(* PLC project SafeLOGIC-1, BrAutomation SafeDESIGNER  4.3.3.7 *)
(* stored: companyURL http://www.br-automation.com, creationDateTime Wed Jan 30 17:54:31 2019 *)

PROGRAM Main
  VAR  (* added by the conversion: wires and edge detectors of the diagram *)
    _AND_S30_OUT : BOOL;
    _AND_S44_OUT : BOOL;
  END_VAR

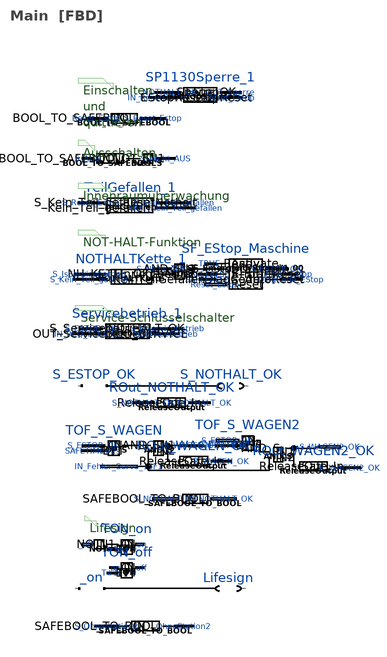
(* FBD diagram, written out as Structured Text *)
(* Einschalten und quittieren *)
SP1130Sperre_1(EStopOK := _NOTHALT_OK, EStopReset := IN_ResetNOTHALT);
Reset_Estop := SP1130Sperre_1.EStopReset2;
OUT_Sperre := SP1130Sperre_1.Sperre;
S_Reset_Estop := BOOL_TO_SAFEBOOL(Reset_Estop);
(* Ausschalten *)
S_Nicht_AUS := NOT_S(BOOL_TO_SAFEBOOL(S_AUS));
(* Innenraumüberwachung *)
TeilGefallen_1(S_ResetNothalt := S_Reset_Estop);
S_Kein_Teil_gefallen := TeilGefallen_1.S_Kein_Teil_gefallen;
OUT_Kein_Teil_gefallen := TeilGefallen_1.Kein_Teil_gefallen;
(* NOT-HALT-Funktion *)
NOTHALTKette_1(Einrichtbetrieb := S_IsServicebetrieb, KeinTeilGefallen := S_Kein_Teil_gefallen);
SF_EStop_Maschine(Activate := TRUE, S_EStopIn := AND_S(S_Nicht_AUS, NOTHALTKette_1.NH_KETTE_OK), S_StartReset := SAFEFALSE, S_AutoReset := SAFEFALSE, Reset := Reset_Estop);
S_ESTOP_OK := SF_EStop_Maschine.S_EStopOut;
DiagCode_EStop := SF_EStop_Maschine.DiagCode;
Error_Estop := SF_EStop_Maschine.Error;
(* Service-Schlüsselschalter *)
Servicebetrieb_1(NOTHALT_OK := S_ESTOP_OK, REQ_SERVICE := IN_REQ_SERVICE);
IsServicebetrieb := Servicebetrieb_1.OUT_Servicebetrieb;
S_IsServicebetrieb := Servicebetrieb_1.S_Servicebetrieb;
S_NOTHALT_OK := S_ESTOP_OK;
ROut_NOTHALT_OK(Safe_In := S_NOTHALT_OK);
R_NOTHALT_OK := ROut_NOTHALT_OK.ReleaseOut;
TOF_S_WAGEN(IN := S_ESTOP_OK, PT := SAFETIME#2s);
_AND_S30_OUT := AND_S(TOF_S_WAGEN.Q, IN_Fehler_Servo_15F1);
S_WAGEN_OK := _AND_S30_OUT;
TOF_S_WAGEN2(IN := S_ESTOP_OK, PT := SAFETIME#2s);
_AND_S44_OUT := AND_S(TOF_S_WAGEN2.Q, IN_Fehler_Servo_15F1);
S_WAGEN2_OK := _AND_S44_OUT;
ROut_WAGEN_OK(Safe_In := _AND_S30_OUT);
R_WAGEN_OK := ROut_WAGEN_OK.ReleaseOut;
ROut_WAGEN2_OK(Safe_In := _AND_S44_OUT);
R_WAGEN2_OK := ROut_WAGEN2_OK.ReleaseOut;
_NOTHALT_OK := SAFEBOOL_TO_BOOL(S_NOTHALT_OK);
(* Lifesign *)
TON_on(IN := NOT _off, PT := T#1s);
_on := TON_on.Q;
TON_off(IN := _on, PT := T#1s);
_off := TON_off.Q;
Lifesign := _on;
OhneStation2 := SAFEBOOL_TO_BOOL(S_OhneStation2);
END_PROGRAM
